TYPE T_GRN_ID :
STRUCT
	Grn: INT;
END_STRUCT
END_TYPE

(* stored: Version 1.1.0.1, ProductVersion 3.1.0.25
   DUT T_GRN_ID: Id {f60abe5f-2361-4659-9b25-9a6949e9a3f5} *)
